// TIA Portal project "Egzamin zawodowy czerwiec 2012 wentylacja" (V11)

(* hardware
DEVICE "S7-400 station_1"  S7400.Device
   slot 0: "UR1_0"  UR1  6ES7 400-1TA01-0AA0
   slot 2: "PLC_1"  CPU 416F-3 PN/DP  6ES7 416-3FR05-0AB0  V5.3
      slot 5: "PROFINET interface_1"  PN-IO
         slot 1: "Port_1"  Port
         slot 2: "Port_2"  Port
*)

// ===== PLC "PLC_1"  CPU 416F-3 PN/DP =====

VAR_GLOBAL   // PLC tag table "Default tag table"
   "S2" AT %I0.1 : Bool;
   "GOTOWOŚĆ" AT %M0.0 : Bool;
   "Tag_1" AT %M1.0 : Bool;
   "S1" AT %I0.0 : Bool;
   "ROZRUCH" AT %M0.1 : Bool;
   "K2 MARKER" AT %M2.0 : Bool;
   "B2" AT %I0.2 : Bool;
   "K1 MARKER" AT %M2.1 : Bool;
   "30 SEKUND" AT %M0.3 : Bool;
   "B1" AT %I0.3 : Bool;
   "POSTÓJ" AT %M0.4 : Bool;
   "PRACA" AT %M0.5 : Bool;
   "LAMPKA" AT %M0.6 : Bool;
   "k1" AT %Q0.0 : Bool;
   "k2" AT %Q0.1 : Bool;
   "lampka(1)" AT %Q0.2 : Bool;
   "Tag_5" AT %M9.7 : Bool;
   "Tag_6" AT %M1.4 : Bool;
   "Tag_7" AT %M7.6 : Bool;
   "Tag_8" AT %M2.2 : Bool;
   "Tag_9" AT %M3.0 : Bool;
   "Tag_10" AT %M4.0 : Bool;
   "Tag_11" AT %M4.4 : Bool;
   "Tag_12" AT %M6.6 : Bool;
END_VAR

ORGANIZATION_BLOCK "Main"   // OB1, LAD
TITLE = "Main Program Sweep (Cycle)"
{ S7_Optimized_Access := 'FALSE' }
VERSION : 0.1
   VAR_TEMP
      OB1_EV_CLASS : Byte;   // Bits 0-3 = 1 (Coming event), Bits 4-7 = 1 (Event class 1)
      OB1_SCAN_1 : Byte;   // 1 (Cold restart scan 1 of OB 1), 3 (Scan 2-n of OB 1)
      OB1_PRIORITY : Byte;   // Priority of OB Execution
      OB1_OB_NUMBR : Byte;   // 1 (Organization block 1, OB1)
      OB1_RESERVED_1 : Byte;   // Reserved for system
      OB1_RESERVED_2 : Byte;   // Reserved for system
      OB1_PREV_CYCLE : Int;   // Cycle time of previous OB1 scan (milliseconds)
      OB1_MIN_CYCLE : Int;   // Minimum cycle time of OB1 (milliseconds)
      OB1_MAX_CYCLE : Int;   // Maximum cycle time of OB1 (milliseconds)
      OB1_DATE_TIME : Date_And_Time;   // Date and time OB1 started
   END_VAR
BEGIN
END_ORGANIZATION_BLOCK